{attribute 'qualified_only'}
VAR_GLOBAL
	rSinValue : REAL;
	aReadStruct : ARRAY[0..200] OF ST_Record;
	
END_VAR

(* stored: Version 1.1.0.1, ProductVersion 3.1.4022.9
   GVL GVL: Id {687bfe43-61b9-4743-a2ed-82a441f30414} *)
